_CFC_ (* Continuous Function Chart, elements in execution order *)
(* 50с *)
#0 AND(TRUE, #11)
#1 YA3_REG_POL <= #0
#2 INT_TO_TIME(SHU6_PV1_YA3_ZADER_RAS_DOST)
#3 MUL(#2, 1000)
#4 TON_YA3_Rassog1:TON(IN: YA3_DOST, PT: #3)
#5 ABS(SHU6_PV1_YA3_RASSOG)
#6 GT(#5, SHU6_PV1_YA3_UST_RASSOG)
#7 AND(NOT SHU6_PV1_UST_RE_PUSK, #12)
#8 GT(SHU6_PV1_YA3_RASSOG, SHU6_PV1_YA3_UST_RASSOG)
#9 SEL(SHU6_PV1_UST_RE_STOP, #6, #8)
#10 ABS(SHU6_PV1_YA3_RASSOG_POL)
#11 GT(#10, SHU6_PV1_YA3_UST_RASSOG)
#12 SEL(YA3_REG_POL, #9, #11)
#13 INT_TO_TIME(SHU6_PV1_YA3_ZADER_RAS)
#14 MUL(#13, 1000)
#15 TON_YA3_Rassog:TON(IN: #7, PT: #14)
#16 OR(#15.Q, YA3_AO_OTKAZ)
#17 AND(#4.Q, SHU6_PV1_1YA3_DI1_A, #16)
#18 SR_YA2_Otk:SR(SET1: #17, RESET: SHU6_PV1_SB)
#19 SHU6_PV1_Z_YA3_OTKAZ <= #18.Q1
_END_CFC_
(* the same logic as Structured Text *)
(* 50с *)
YA3_REG_POL := TRUE AND _t14;
TON_YA3_Rassog1(IN := YA3_DOST, PT := INT_TO_TIME(SHU6_PV1_YA3_ZADER_RAS_DOST) * 1000);
_t140 := NOT SHU6_PV1_UST_RE_PUSK AND _t84;
_t14 := ABS(SHU6_PV1_YA3_RASSOG_POL) > SHU6_PV1_YA3_UST_RASSOG;
_t84 := SEL(YA3_REG_POL, SEL(SHU6_PV1_UST_RE_STOP, ABS(SHU6_PV1_YA3_RASSOG) > SHU6_PV1_YA3_UST_RASSOG, SHU6_PV1_YA3_RASSOG > SHU6_PV1_YA3_UST_RASSOG), _t14);
TON_YA3_Rassog(IN := _t140, PT := INT_TO_TIME(SHU6_PV1_YA3_ZADER_RAS) * 1000);
SR_YA2_Otk(SET1 := TON_YA3_Rassog1.Q AND SHU6_PV1_1YA3_DI1_A AND (TON_YA3_Rassog.Q OR YA3_AO_OTKAZ), RESET := SHU6_PV1_SB);
SHU6_PV1_Z_YA3_OTKAZ := SR_YA2_Otk.Q1;
END_PROGRAM

(* POU TZBiS/TZB/Z_YA4_Otk, CFC *)
PROGRAM Z_YA4_Otk
VAR
	SR_YA4_Otk: SR;
	TON_YA4_Zakl: TON;
END_VAR
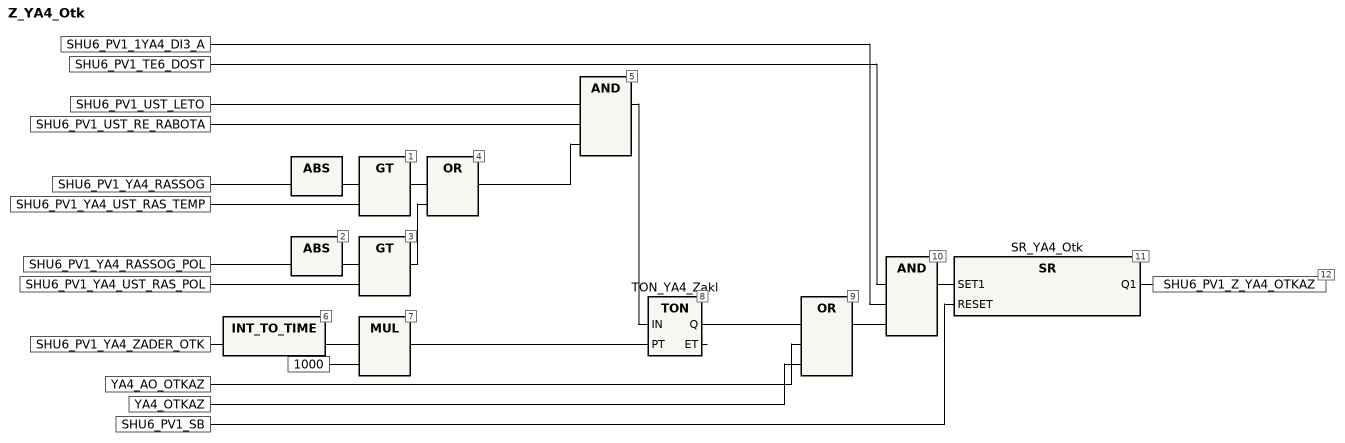
_CFC_ (* Continuous Function Chart, elements in execution order *)
#0 ABS(SHU6_PV1_YA4_RASSOG)
#1 GT(#0, SHU6_PV1_YA4_UST_RAS_TEMP)
#2 ABS(SHU6_PV1_YA4_RASSOG_POL)
#3 GT(#2, SHU6_PV1_YA4_UST_RAS_POL)
#4 OR(#1, #3)
#5 AND(SHU6_PV1_UST_LETO, SHU6_PV1_UST_RE_RABOTA, #4)
#6 INT_TO_TIME(SHU6_PV1_YA4_ZADER_OTK)
#7 MUL(#6, 1000)
#8 TON_YA4_Zakl:TON(IN: #5, PT: #7)
#9 OR(#8.Q, YA4_AO_OTKAZ, YA4_OTKAZ)
#10 AND(SHU6_PV1_TE6_DOST, SHU6_PV1_1YA4_DI3_A, #9)
#11 SR_YA4_Otk:SR(SET1: #10, RESET: SHU6_PV1_SB)
#12 SHU6_PV1_Z_YA4_OTKAZ <= #11.Q1
_END_CFC_
(* the same logic as Structured Text *)
TON_YA4_Zakl(IN := SHU6_PV1_UST_LETO AND SHU6_PV1_UST_RE_RABOTA AND ((ABS(SHU6_PV1_YA4_RASSOG) > SHU6_PV1_YA4_UST_RAS_TEMP) OR (ABS(SHU6_PV1_YA4_RASSOG_POL) > SHU6_PV1_YA4_UST_RAS_POL)), PT := INT_TO_TIME(SHU6_PV1_YA4_ZADER_OTK) * 1000);
SR_YA4_Otk(SET1 := SHU6_PV1_TE6_DOST AND SHU6_PV1_1YA4_DI3_A AND (TON_YA4_Zakl.Q OR YA4_AO_OTKAZ OR YA4_OTKAZ), RESET := SHU6_PV1_SB);
SHU6_PV1_Z_YA4_OTKAZ := SR_YA4_Otk.Q1;
END_PROGRAM

(* POU TZBiS/TZB/Z_Zam, CFC *)
PROGRAM Z_Zam
VAR
	RT_VKL: R_TRIG;
	SR_ZAM: SR;
	TON_VKL: TON;
	TP_VKL: TON;
	FT_TP_VKL: F_TRIG;
	SR_TS: SR;
END_VAR
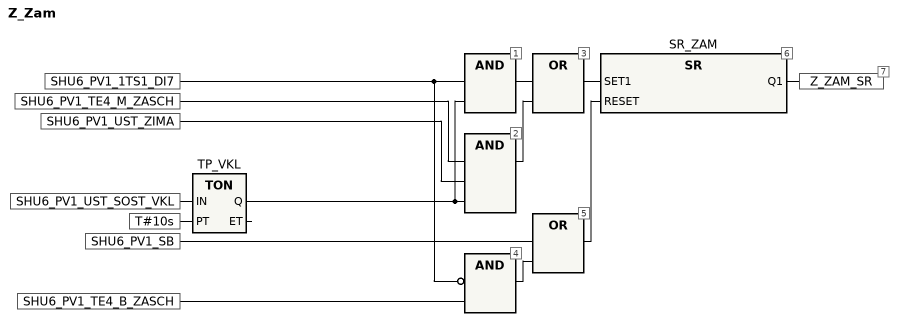
_CFC_ (* Continuous Function Chart, elements in execution order *)
#0 TP_VKL:TON(IN: SHU6_PV1_UST_SOST_VKL, PT: T#10s)
#1 AND(SHU6_PV1_1TS1_DI7, #0.Q)
#2 AND(SHU6_PV1_TE4_M_ZASCH, SHU6_PV1_UST_ZIMA, #0.Q)
#3 OR(#1, #2)
#4 AND(NOT SHU6_PV1_1TS1_DI7, SHU6_PV1_TE4_B_ZASCH)
#5 OR(SHU6_PV1_SB, #4)
#6 SR_ZAM:SR(SET1: #3, RESET: #5)
#7 Z_ZAM_SR <= #6.Q1
_END_CFC_
(* the same logic as Structured Text *)
TP_VKL(IN := SHU6_PV1_UST_SOST_VKL, PT := T#10s);
SR_ZAM(SET1 := (SHU6_PV1_1TS1_DI7 AND TP_VKL.Q) OR (SHU6_PV1_TE4_M_ZASCH AND SHU6_PV1_UST_ZIMA AND TP_VKL.Q), RESET := SHU6_PV1_SB OR (NOT SHU6_PV1_1TS1_DI7 AND SHU6_PV1_TE4_B_ZASCH));
Z_ZAM_SR := SR_ZAM.Q1;
END_PROGRAM

(* POU TZBiS/TZB/Z_Dlit_Ster_Reg, CFC *)
	PROGRAM Z_Dlit_Ster_Reg
VAR
	SR_HZ20S60: SR;
	LT_HZm20: ISTOK_LT;
	TON_HZm20: TON;
END_VAR
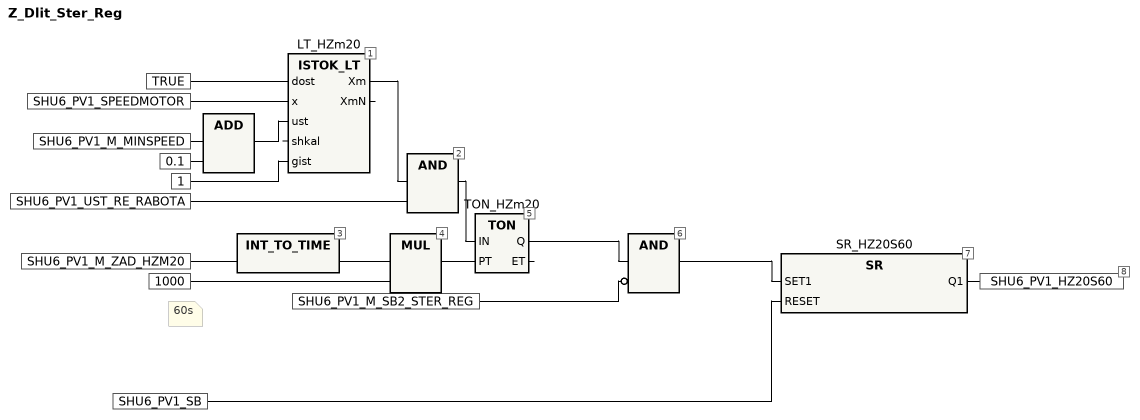
_CFC_ (* Continuous Function Chart, elements in execution order *)
(* 60s *)
#0 ADD(SHU6_PV1_M_MINSPEED, 0.1)
#1 LT_HZm20:ISTOK_LT(dost: TRUE, x: SHU6_PV1_SPEEDMOTOR, ust: #0, shkal: -, gist: 1)
#2 AND(#1.Xm, SHU6_PV1_UST_RE_RABOTA)
#3 INT_TO_TIME(SHU6_PV1_M_ZAD_HZM20)
#4 MUL(#3, 1000)
#5 TON_HZm20:TON(IN: #2, PT: #4)
#6 AND(#5.Q, NOT SHU6_PV1_M_SB2_STER_REG)
#7 SR_HZ20S60:SR(SET1: #6, RESET: SHU6_PV1_SB)
#8 SHU6_PV1_HZ20S60 <= #7.Q1
_END_CFC_
(* the same logic as Structured Text *)
(* 60s *)
LT_HZm20(dost := TRUE, x := SHU6_PV1_SPEEDMOTOR, ust := SHU6_PV1_M_MINSPEED + 0.1, gist := 1);
TON_HZm20(IN := LT_HZm20.Xm AND SHU6_PV1_UST_RE_RABOTA, PT := INT_TO_TIME(SHU6_PV1_M_ZAD_HZM20) * 1000);
SR_HZ20S60(SET1 := TON_HZm20.Q AND NOT SHU6_PV1_M_SB2_STER_REG, RESET := SHU6_PV1_SB);
SHU6_PV1_HZ20S60 := SR_HZ20S60.Q1;
END_PROGRAM

(* POU TZBiS/TZB/Z_ALL, CFC *)
PROGRAM Z_ALL
VAR
	SR_Z_all: SR;
END_VAR
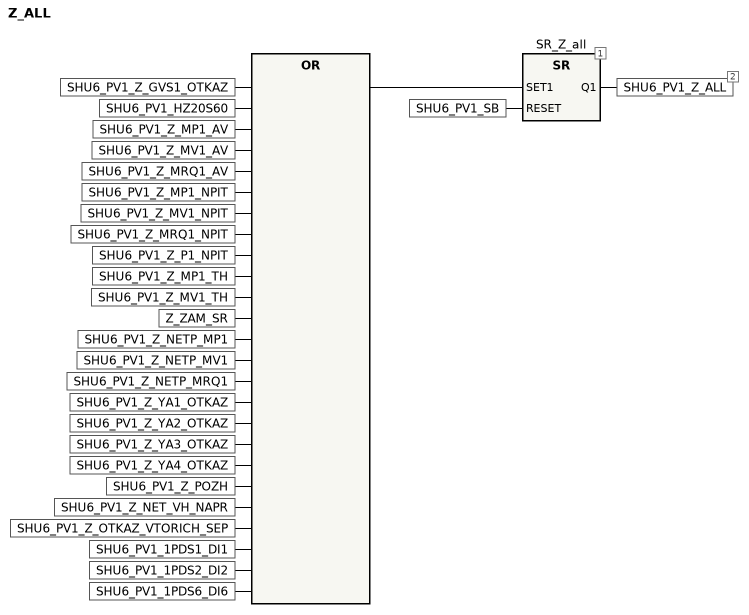
_CFC_ (* Continuous Function Chart, elements in execution order *)
#0 OR(SHU6_PV1_Z_GVS1_OTKAZ, SHU6_PV1_HZ20S60, SHU6_PV1_Z_MP1_AV, SHU6_PV1_Z_MV1_AV, SHU6_PV1_Z_MRQ1_AV, SHU6_PV1_Z_MP1_NPIT, SHU6_PV1_Z_MV1_NPIT, SHU6_PV1_Z_MRQ1_NPIT, SHU6_PV1_Z_P1_NPIT, SHU6_PV1_Z_MP1_TH, SHU6_PV1_Z_MV1_TH, Z_ZAM_SR, SHU6_PV1_Z_NETP_MP1, SHU6_PV1_Z_NETP_MV1, SHU6_PV1_Z_NETP_MRQ1, SHU6_PV1_Z_YA1_OTKAZ, SHU6_PV1_Z_YA2_OTKAZ, SHU6_PV1_Z_YA3_OTKAZ, SHU6_PV1_Z_YA4_OTKAZ, SHU6_PV1_Z_POZH, SHU6_PV1_Z_NET_VH_NAPR, SHU6_PV1_Z_OTKAZ_VTORICH_SEP, SHU6_PV1_1PDS1_DI1, SHU6_PV1_1PDS2_DI2, SHU6_PV1_1PDS6_DI6)
#1 SR_Z_all:SR(SET1: #0, RESET: SHU6_PV1_SB)
#2 SHU6_PV1_Z_ALL <= #1.Q1
_END_CFC_
(* the same logic as Structured Text *)
SR_Z_all(SET1 := SHU6_PV1_Z_GVS1_OTKAZ OR SHU6_PV1_HZ20S60 OR SHU6_PV1_Z_MP1_AV OR SHU6_PV1_Z_MV1_AV OR SHU6_PV1_Z_MRQ1_AV OR SHU6_PV1_Z_MP1_NPIT OR SHU6_PV1_Z_MV1_NPIT OR SHU6_PV1_Z_MRQ1_NPIT OR SHU6_PV1_Z_P1_NPIT OR SHU6_PV1_Z_MP1_TH OR SHU6_PV1_Z_MV1_TH OR Z_ZAM_SR OR SHU6_PV1_Z_NETP_MP1 OR SHU6_PV1_Z_NETP_MV1 OR SHU6_PV1_Z_NETP_MRQ1 OR SHU6_PV1_Z_YA1_OTKAZ OR SHU6_PV1_Z_YA2_OTKAZ OR SHU6_PV1_Z_YA3_OTKAZ OR SHU6_PV1_Z_YA4_OTKAZ OR SHU6_PV1_Z_POZH OR SHU6_PV1_Z_NET_VH_NAPR OR SHU6_PV1_Z_OTKAZ_VTORICH_SEP OR SHU6_PV1_1PDS1_DI1 OR SHU6_PV1_1PDS2_DI2 OR SHU6_PV1_1PDS6_DI6, RESET := SHU6_PV1_SB);
SHU6_PV1_Z_ALL := SR_Z_all.Q1;
END_PROGRAM

(* POU Regim/ALL_Regim, CFC *)
PROGRAM ALL_Regim
VAR
END_VAR
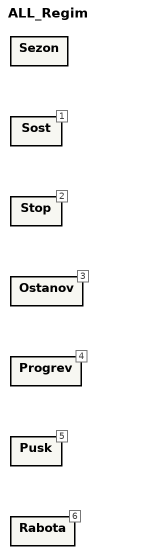
_CFC_ (* Continuous Function Chart, elements in execution order *)
#0 Sezon()
#1 Sost()
#2 Stop()
#3 Ostanov()
#4 Progrev()
#5 Pusk()
#6 Rabota()
_END_CFC_
(* the same logic as Structured Text *)
Sezon();
Sost();
Stop();
Ostanov();
Progrev();
Pusk();
Rabota();
END_PROGRAM

(* POU Regim/Sezon, CFC *)
PROGRAM Sezon
VAR
	RS_Sezon: RS;
	RT_Zima: R_TRIG;
	RT_Leto: R_TRIG;
	RT_Auto: R_TRIG;
	RS_Auto: RS;
	RT_T: R_TRIG;
END_VAR
VAR (* helpers for the ST form of the networks *)
	_t72 : BOOL;
END_VAR
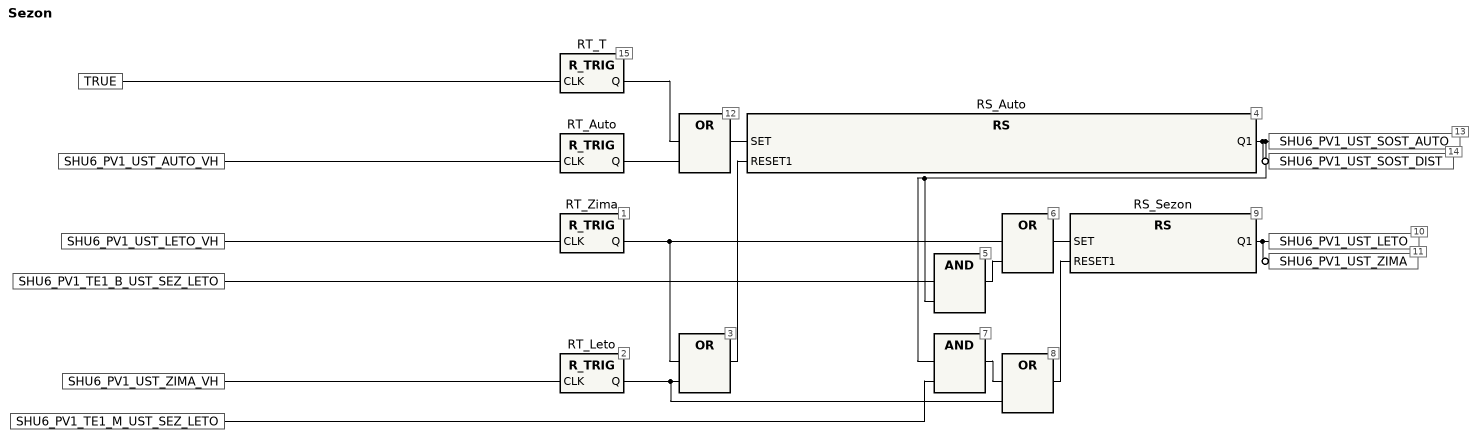
_CFC_ (* Continuous Function Chart, elements in execution order *)
#0 RT_Auto:R_TRIG(CLK: SHU6_PV1_UST_AUTO_VH)
#1 RT_Zima:R_TRIG(CLK: SHU6_PV1_UST_LETO_VH)
#2 RT_Leto:R_TRIG(CLK: SHU6_PV1_UST_ZIMA_VH)
#3 OR(#1.Q, #2.Q)
#4 RS_Auto:RS(SET: #12, RESET1: #3)
#5 AND(SHU6_PV1_TE1_B_UST_SEZ_LETO, #4.Q1)
#6 OR(#1.Q, #5)
#7 AND(#4.Q1, SHU6_PV1_TE1_M_UST_SEZ_LETO)
#8 OR(#7, #2.Q)
#9 RS_Sezon:RS(SET: #6, RESET1: #8)
#10 SHU6_PV1_UST_LETO <= #9.Q1
#11 SHU6_PV1_UST_ZIMA <= NOT #9.Q1
#12 OR(#15.Q, #0.Q)
#13 SHU6_PV1_UST_SOST_AUTO <= #4.Q1
#14 SHU6_PV1_UST_SOST_DIST <= NOT #4.Q1
#15 RT_T:R_TRIG(CLK: TRUE)
_END_CFC_
(* the same logic as Structured Text *)
RT_Auto(CLK := SHU6_PV1_UST_AUTO_VH);
RT_Zima(CLK := SHU6_PV1_UST_LETO_VH);
RT_Leto(CLK := SHU6_PV1_UST_ZIMA_VH);
RS_Auto(SET := _t72, RESET1 := RT_Zima.Q OR RT_Leto.Q);
RS_Sezon(SET := RT_Zima.Q OR (SHU6_PV1_TE1_B_UST_SEZ_LETO AND RS_Auto.Q1), RESET1 := (RS_Auto.Q1 AND SHU6_PV1_TE1_M_UST_SEZ_LETO) OR RT_Leto.Q);
SHU6_PV1_UST_LETO := RS_Sezon.Q1;
SHU6_PV1_UST_ZIMA := NOT RS_Sezon.Q1;
_t72 := RT_T.Q OR RT_Auto.Q;
SHU6_PV1_UST_SOST_AUTO := RS_Auto.Q1;
SHU6_PV1_UST_SOST_DIST := NOT RS_Auto.Q1;
RT_T(CLK := TRUE);
END_PROGRAM

(* POU Regim/Sost, CFC *)
PROGRAM Sost
VAR
	RS_Sost: RS;
	RT_PUSK: R_TRIG;
	RT_STOP: R_TRIG;
	RS_Old_Sost: RS;
	TON_Kv1: TON;
	TON_Kv1_1: TON;
	OLD_SOST: BOOL;

	KV1: BOOL;
	RT_PUSK_OLD: R_TRIG;
	CTU_TS: CTU;
	TOF_TS_1: TOF;
	TOF_TS_2: TOF;
	TOF_TS_3: TOF;
	RT_PUSK_OLD1: R_TRIG;
	TON_Kv1_11: TON;
	TON_Kv11: TON;
	TOF_TE_1: TOF;
	TOF_Te_2: TOF;
	TOF_Te_3: TOF;
	CTU_Te: CTU;
END_VAR
